_CFC_ (* Continuous Function Chart, elements in execution order *)
#0 AND(SHU6_PV1_UST_RE_PUSK, NOT SHU6_PV1_YA1_DI3_ZKR)
#1 mv_1_TON:TON(IN: #0, PT: t#6s)
#2 OR(#1.Q, SHU6_PV1_UST_RE_RABOTA)
#3 OR(SHU6_PV1_UST_RE_OSTANOV, SHU6_PV1_UST_RE_STOP)
#4 SR_VKL:SR(SET1: #2, RESET: #3)
#5 OR(SHU6_PV1_Z_MV1_TH, SHU6_PV1_MV1_DI2_ALM, SHU6_PV1_Z_MV1_NPIT)
#6 AND(SHU6_PV1_YAMV1_DI7_A, SHU6_PV1_MV1_DI2_RUN)
#7 fb_HVACMS_M2:FB_HVACMotor1Speed(eHVACDataSecurityType_Idle, FALSE, TRUE, #4.Q1, eHVACActuatorMode_Auto_BMS, NOT #5, #6, NOT SHU6_PV1_Z_NETP_MV1, TRUE, TRUE, TRUE, SHU6_PV1_SB, startDelay_M2, stopDelay_M2, delayFBC_M2, feedbPT_M2, delayFBP_M2)
#8 SHU6_PV1_MV1_DO3_VKL <= #7.out 1
#9 MV1_OTKAZ <= #7.out 7
#10 INT_TO_TIME(SHU6_PV1_M_TI)
#11 MUL(#10, 1000)
#12 tTi <= #11
_END_CFC_
END_PROGRAM

(* POU IM/CHASTOTA_M1_M2, CFC *)
PROGRAM CHASTOTA_M1_M2
VAR
	RR: RAMP_REAL;
	SR_START_STER_REG: SR;
	SR_START_POV_REG: RS;
	RT_KOMVKL: R_TRIG;
	RT_KOMVKL_2: R_TRIG;
	RT_KOMVKL_1: R_TRIG;
	Zad_PE: TON;
	RS_RUCH: RS;
	V_RUCH: BOOL;
	TON_RUCH: TON;
	SHU6_PV1_M_MAXSPEED_CH_OLD: REAL;
	TON_STER_1: TON;
	TON_STER_2: TON;
	RT_PDK: R_TRIG;
	FT_PDK: F_TRIG;
	RT_KOMVKL_3: R_TRIG;
END_VAR
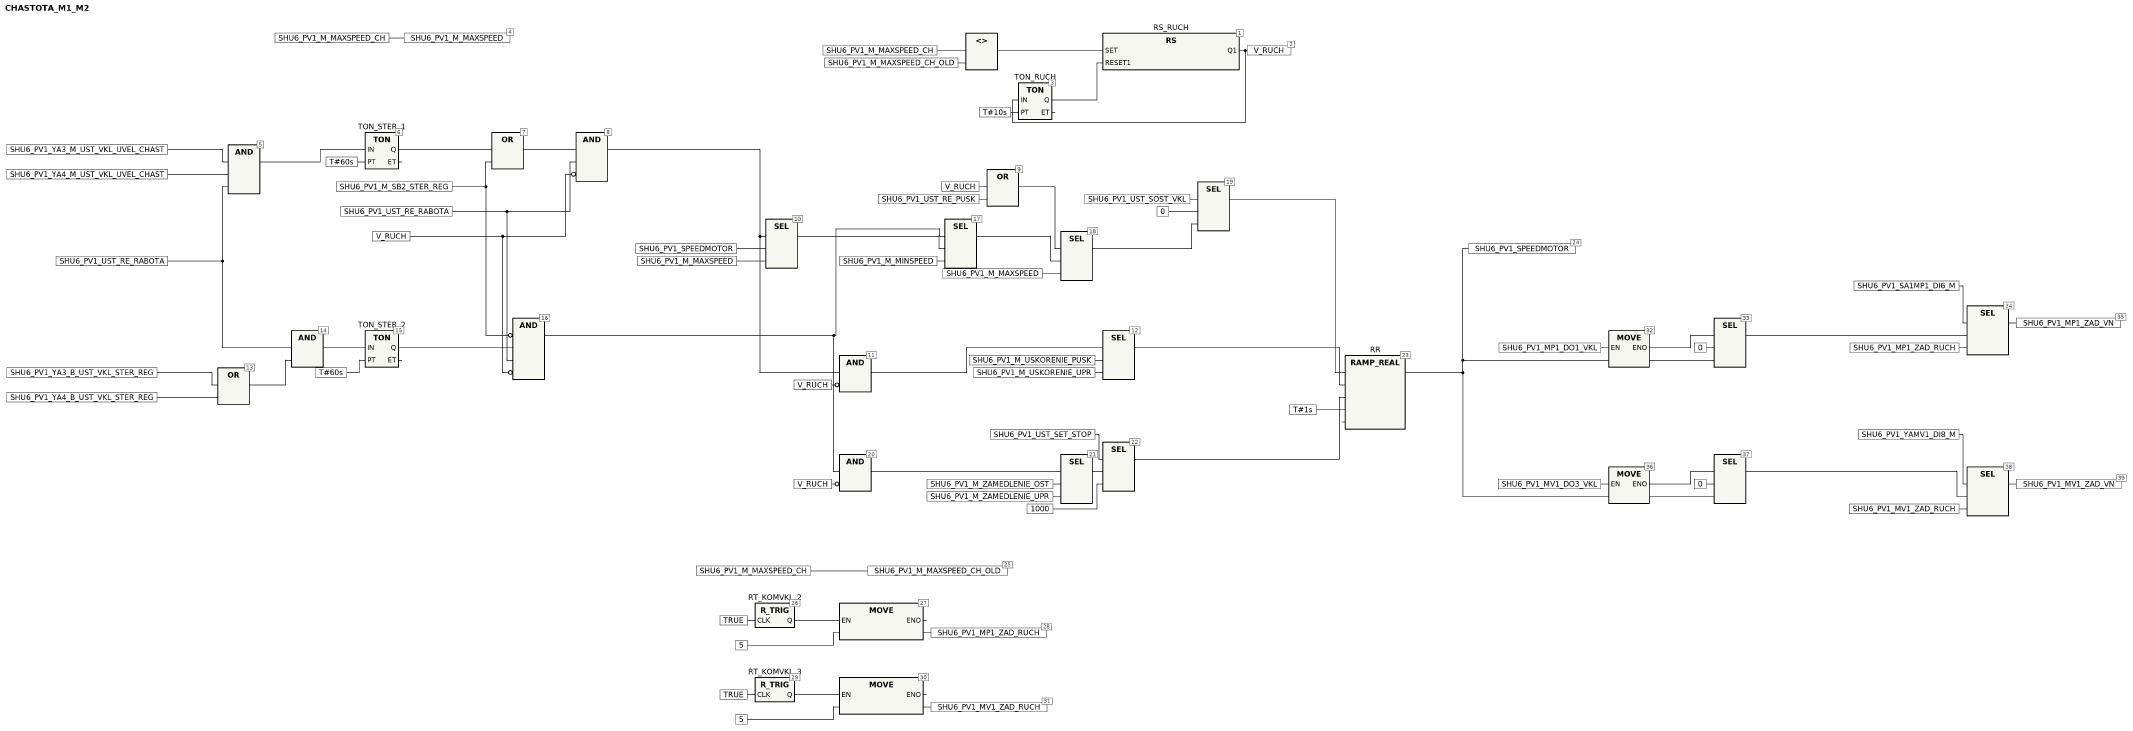
